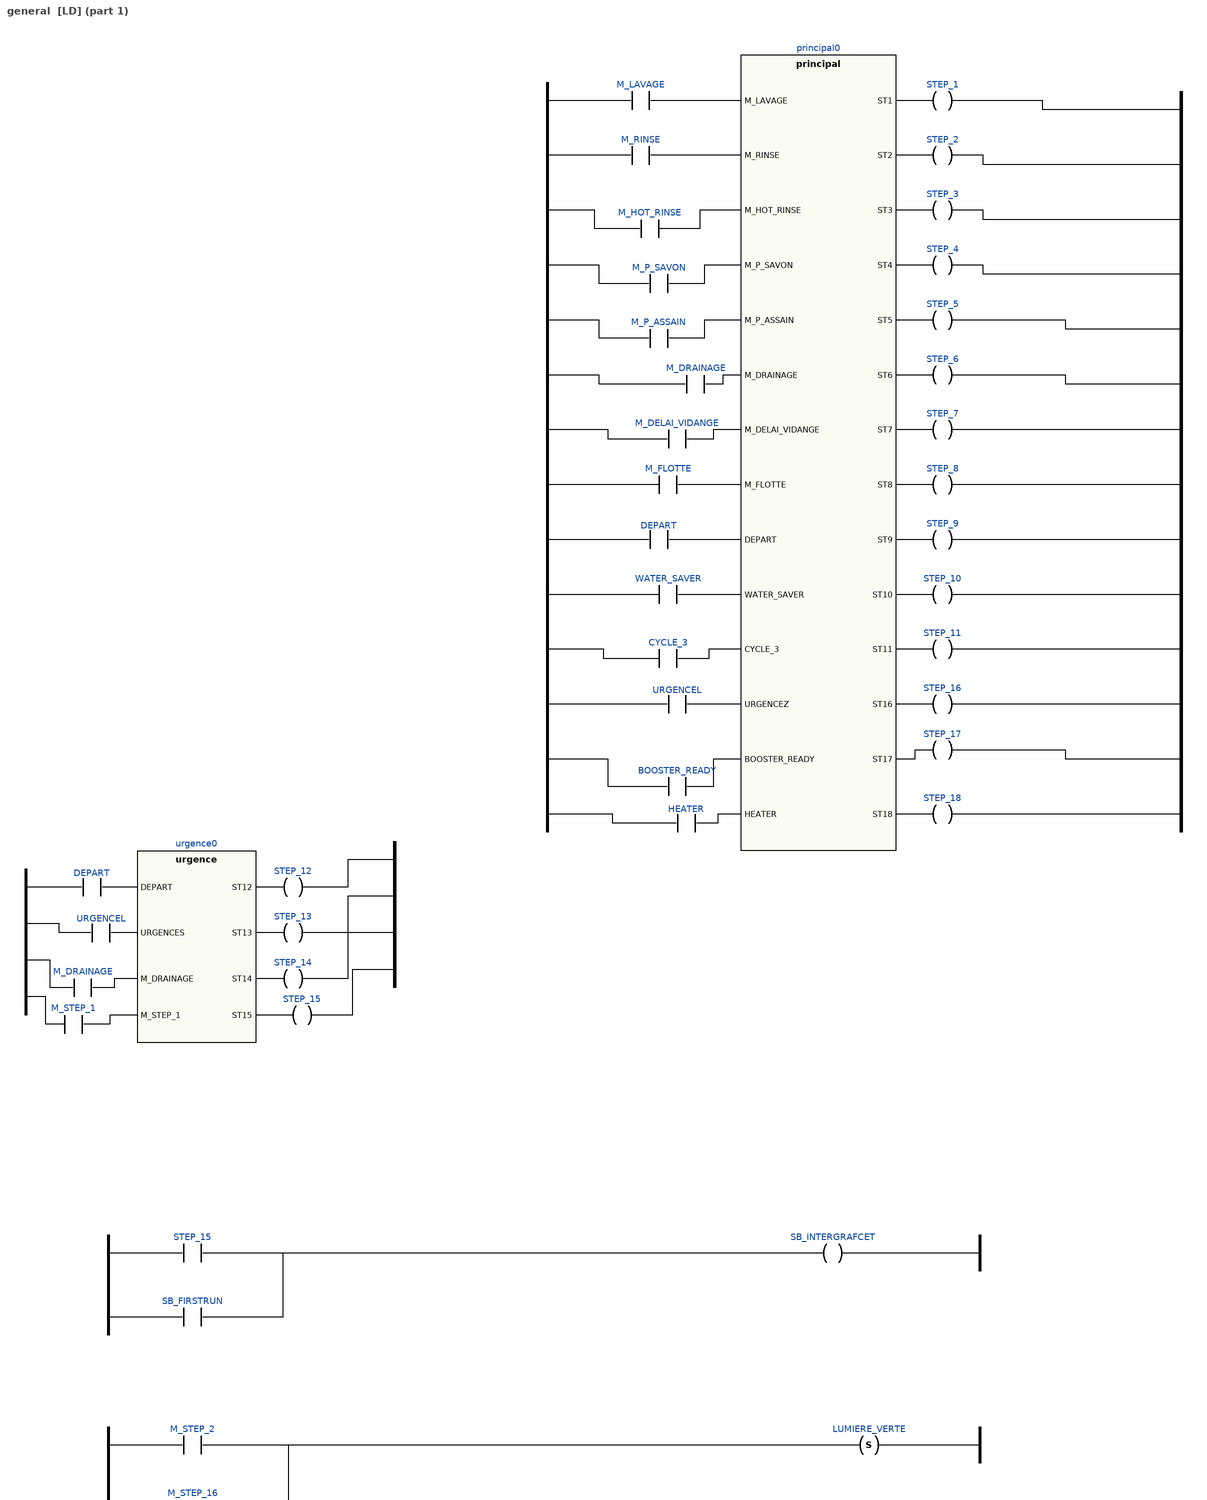
(* LD diagram, written out as Structured Text *)
principal0(M_LAVAGE := M_LAVAGE, M_RINSE := M_RINSE, M_HOT_RINSE := M_HOT_RINSE, M_P_SAVON := M_P_SAVON, M_P_ASSAIN := M_P_ASSAIN, M_DRAINAGE := M_DRAINAGE, M_DELAI_VIDANGE := M_DELAI_VIDANGE, M_FLOTTE := M_FLOTTE, DEPART := DEPART, WATER_SAVER := WATER_SAVER, CYCLE_3 := CYCLE_3, URGENCEZ := URGENCEL, BOOSTER_READY := BOOSTER_READY, HEATER := HEATER);
STEP_1 := principal0.ST1;
STEP_2 := principal0.ST2;
STEP_3 := principal0.ST3;
STEP_4 := principal0.ST4;
STEP_5 := principal0.ST5;
STEP_6 := principal0.ST6;
STEP_7 := principal0.ST7;
STEP_8 := principal0.ST8;
STEP_9 := principal0.ST9;
STEP_10 := principal0.ST10;
STEP_11 := principal0.ST11;
STEP_16 := principal0.ST16;
STEP_17 := principal0.ST17;
STEP_18 := principal0.ST18;
urgence0(DEPART := DEPART, URGENCES := URGENCEL, M_DRAINAGE := M_DRAINAGE, M_STEP_1 := M_STEP_1);
STEP_12 := urgence0.ST12;
STEP_13 := urgence0.ST13;
STEP_14 := urgence0.ST14;
STEP_15 := urgence0.ST15;
SB_INTERGRAFCET := STEP_15 OR SB_FIRSTRUN;
IF M_STEP_2 OR M_STEP_16 THEN LUMIERE_VERTE := TRUE; END_IF;
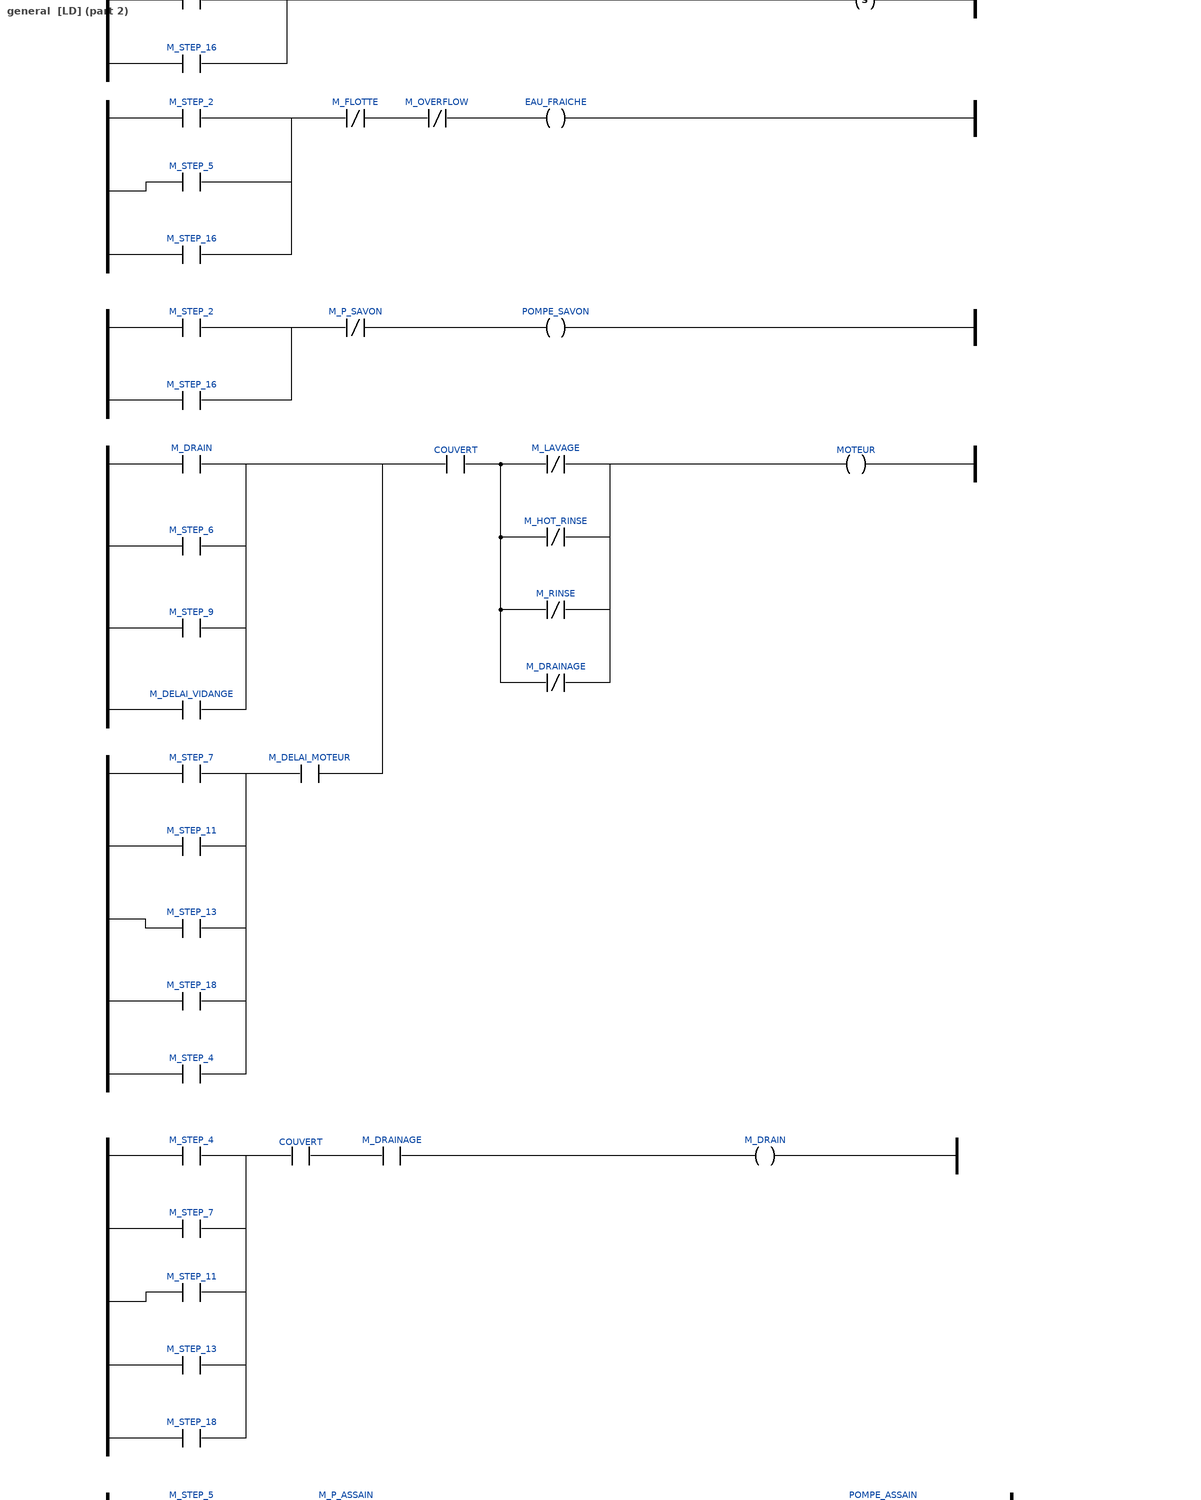
EAU_FRAICHE := (M_STEP_2 OR M_STEP_5 OR M_STEP_16) AND NOT M_FLOTTE AND NOT M_OVERFLOW;
POMPE_SAVON := (M_STEP_2 OR M_STEP_16) AND NOT M_P_SAVON;
MOTEUR := (M_DRAIN OR M_STEP_6 OR M_STEP_9 OR M_DELAI_VIDANGE OR (M_STEP_7 OR M_STEP_11 OR M_STEP_13 OR M_STEP_18 OR M_STEP_4) AND M_DELAI_MOTEUR) AND COUVERT AND (NOT M_LAVAGE OR NOT M_HOT_RINSE OR NOT M_RINSE OR NOT M_DRAINAGE);
M_DRAIN := (M_STEP_4 OR M_STEP_7 OR M_STEP_11 OR M_STEP_13 OR M_STEP_18) AND COUVERT AND M_DRAINAGE;
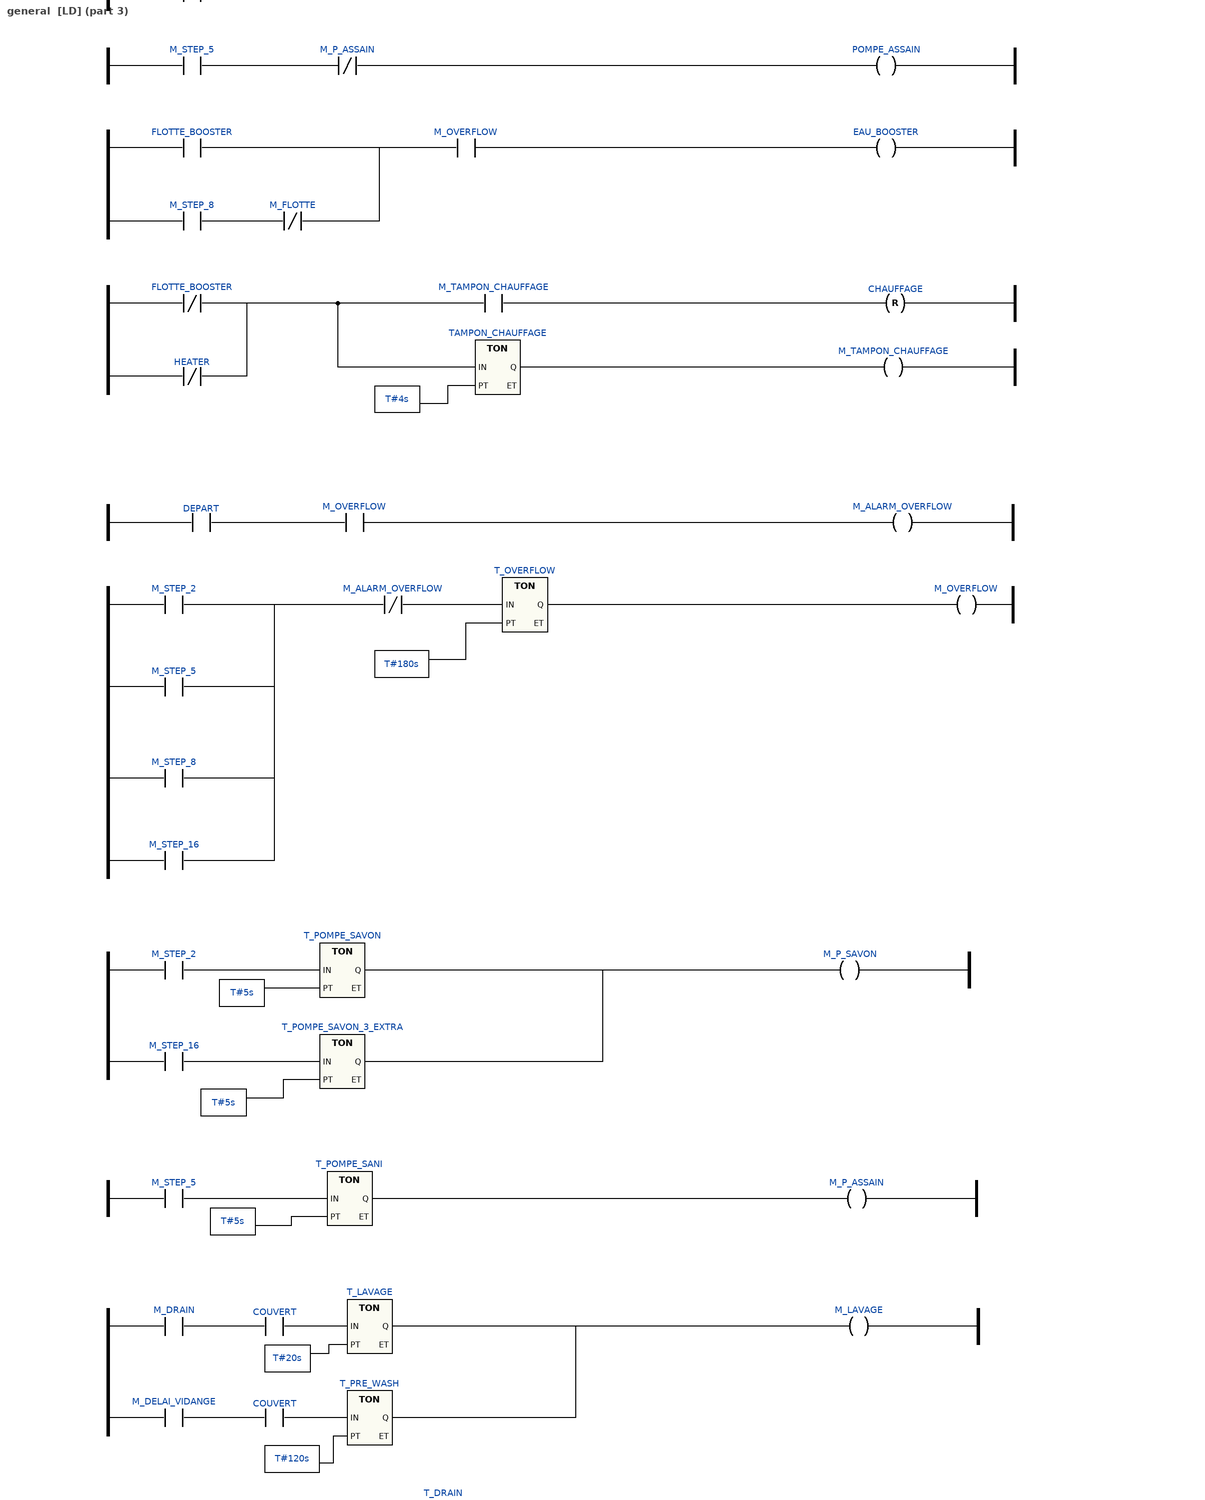
POMPE_ASSAIN := M_STEP_5 AND NOT M_P_ASSAIN;
EAU_BOOSTER := (M_STEP_8 AND NOT M_FLOTTE OR FLOTTE_BOOSTER) AND M_OVERFLOW;
IF (NOT FLOTTE_BOOSTER OR NOT HEATER) AND M_TAMPON_CHAUFFAGE THEN CHAUFFAGE := FALSE; END_IF;
TAMPON_CHAUFFAGE(IN := NOT FLOTTE_BOOSTER, PT := T#4s);
M_TAMPON_CHAUFFAGE := TAMPON_CHAUFFAGE.Q;
M_ALARM_OVERFLOW := DEPART AND M_OVERFLOW;
T_OVERFLOW(IN := (M_STEP_2 OR M_STEP_5 OR M_STEP_8 OR M_STEP_16) AND NOT M_ALARM_OVERFLOW, PT := T#180s);
M_OVERFLOW := T_OVERFLOW.Q;
T_POMPE_SAVON(IN := M_STEP_2, PT := T#5s);
T_POMPE_SAVON_3_EXTRA(IN := M_STEP_16, PT := T#5s);
M_P_SAVON := T_POMPE_SAVON.Q OR T_POMPE_SAVON_3_EXTRA.Q;
T_POMPE_SANI(IN := M_STEP_5, PT := T#5s);
M_P_ASSAIN := T_POMPE_SANI.Q;
T_LAVAGE(IN := M_DRAIN AND COUVERT, PT := T#20s);
T_PRE_WASH(IN := M_DELAI_VIDANGE AND COUVERT, PT := T#120s);
M_LAVAGE := T_LAVAGE.Q OR T_PRE_WASH.Q;
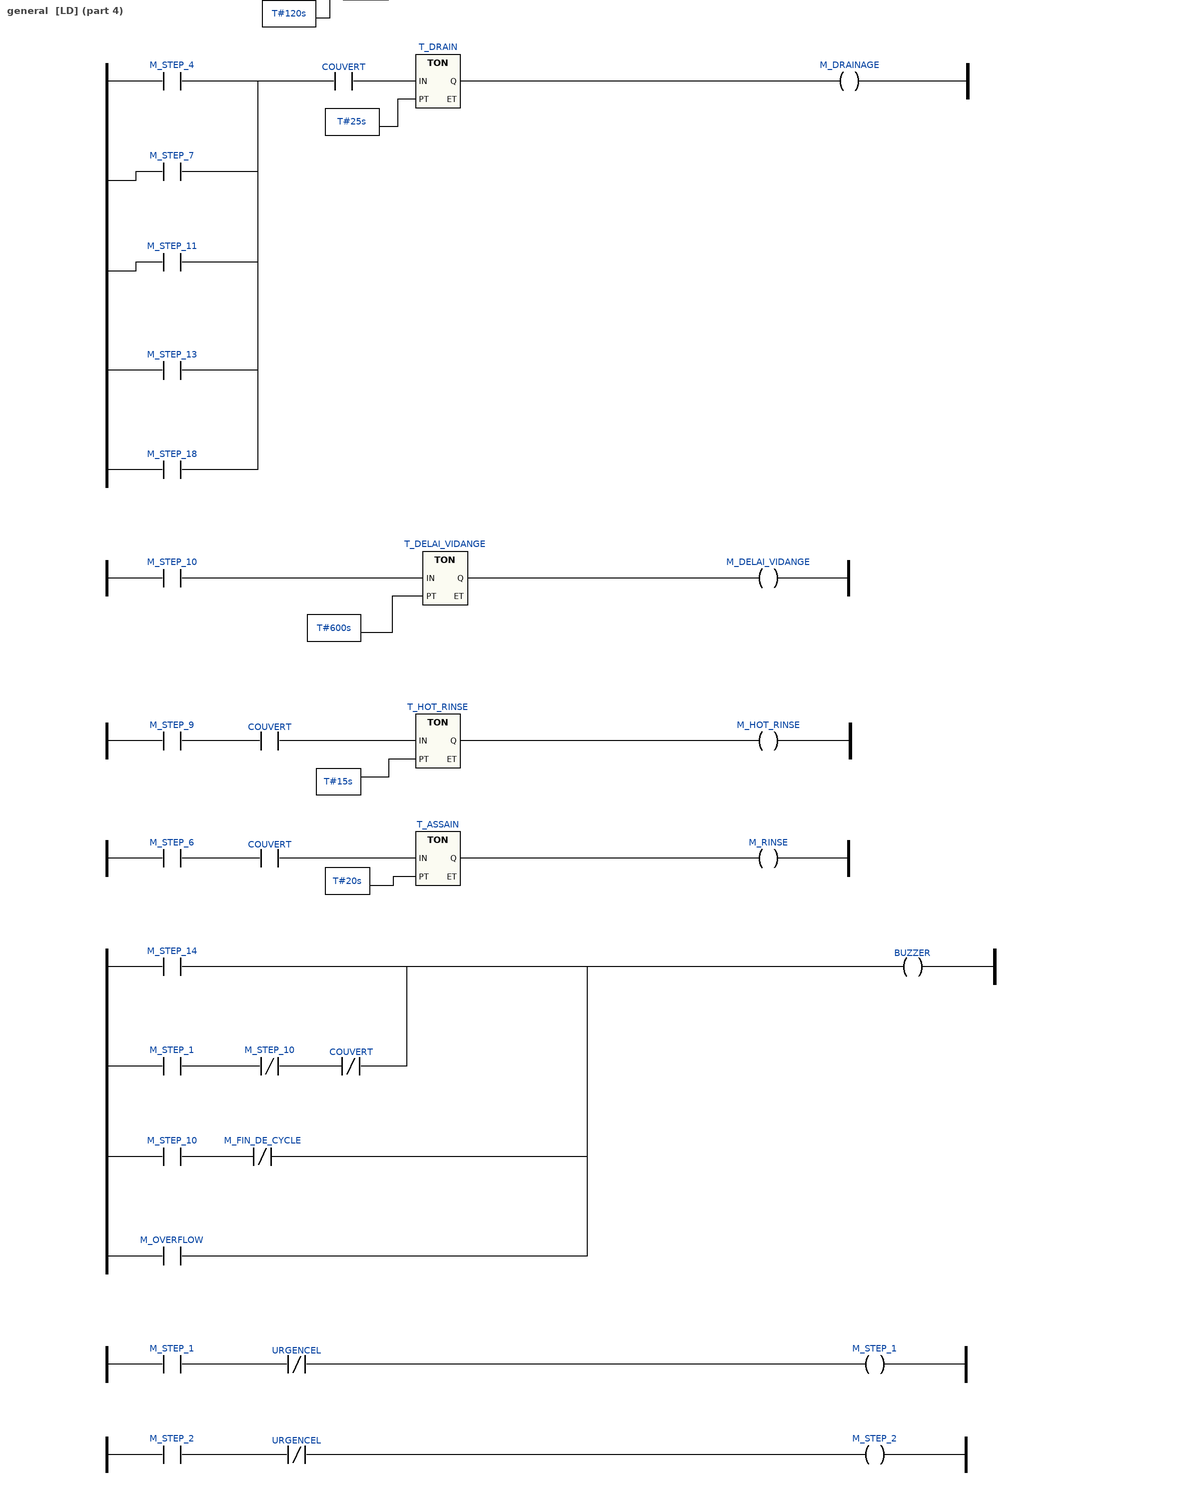
T_DRAIN(IN := (M_STEP_4 OR M_STEP_7 OR M_STEP_11 OR M_STEP_13 OR M_STEP_18) AND COUVERT, PT := T#25s);
M_DRAINAGE := T_DRAIN.Q;
T_DELAI_VIDANGE(IN := M_STEP_10, PT := T#600s);
M_DELAI_VIDANGE := T_DELAI_VIDANGE.Q;
T_HOT_RINSE(IN := M_STEP_9 AND COUVERT, PT := T#15s);
M_HOT_RINSE := T_HOT_RINSE.Q;
T_ASSAIN(IN := M_STEP_6 AND COUVERT, PT := T#20s);
M_RINSE := T_ASSAIN.Q;
BUZZER := M_STEP_14 OR M_STEP_1 AND NOT M_STEP_10 AND NOT COUVERT OR M_STEP_10 AND NOT M_FIN_DE_CYCLE OR M_OVERFLOW;
M_STEP_1 := M_STEP_1 AND NOT URGENCEL;
M_STEP_2 := M_STEP_2 AND NOT URGENCEL;
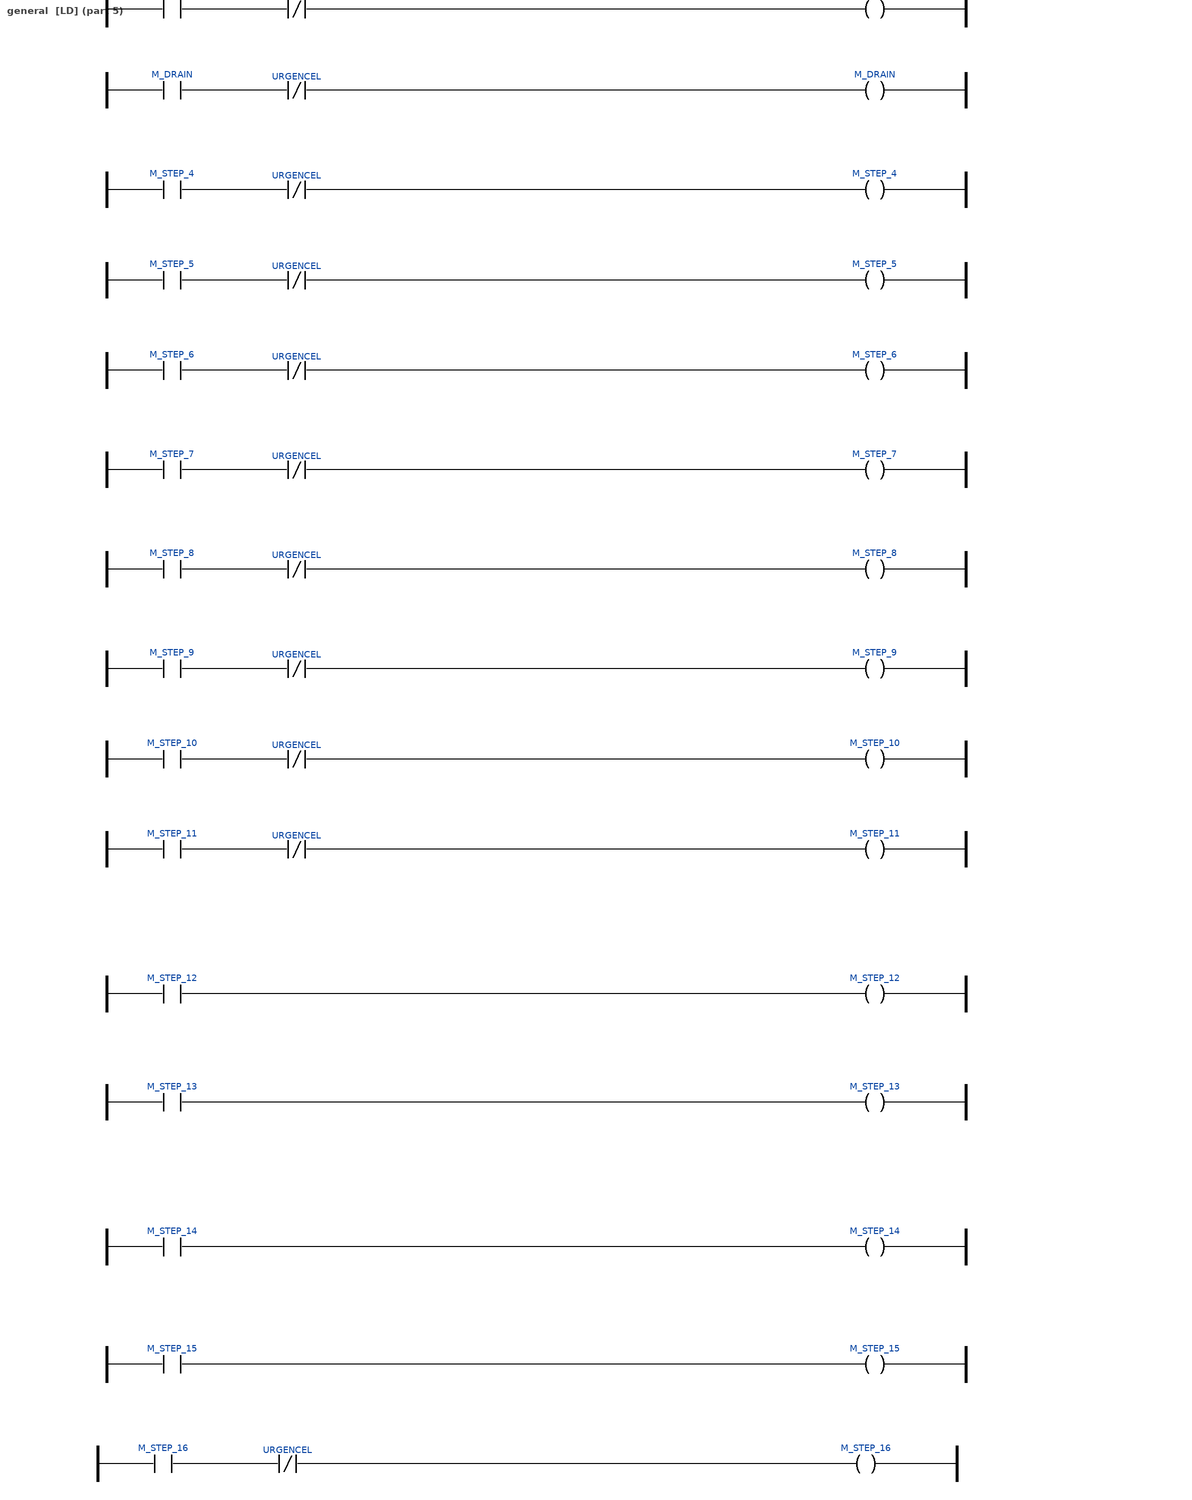
M_DRAIN := M_DRAIN AND NOT URGENCEL;
M_STEP_4 := M_STEP_4 AND NOT URGENCEL;
M_STEP_5 := M_STEP_5 AND NOT URGENCEL;
M_STEP_6 := M_STEP_6 AND NOT URGENCEL;
M_STEP_7 := M_STEP_7 AND NOT URGENCEL;
M_STEP_8 := M_STEP_8 AND NOT URGENCEL;
M_STEP_9 := M_STEP_9 AND NOT URGENCEL;
M_STEP_10 := M_STEP_10 AND NOT URGENCEL;
M_STEP_11 := M_STEP_11 AND NOT URGENCEL;
M_STEP_12 := M_STEP_12;
M_STEP_13 := M_STEP_13;
M_STEP_14 := M_STEP_14;
M_STEP_15 := M_STEP_15;
M_STEP_16 := M_STEP_16 AND NOT URGENCEL;
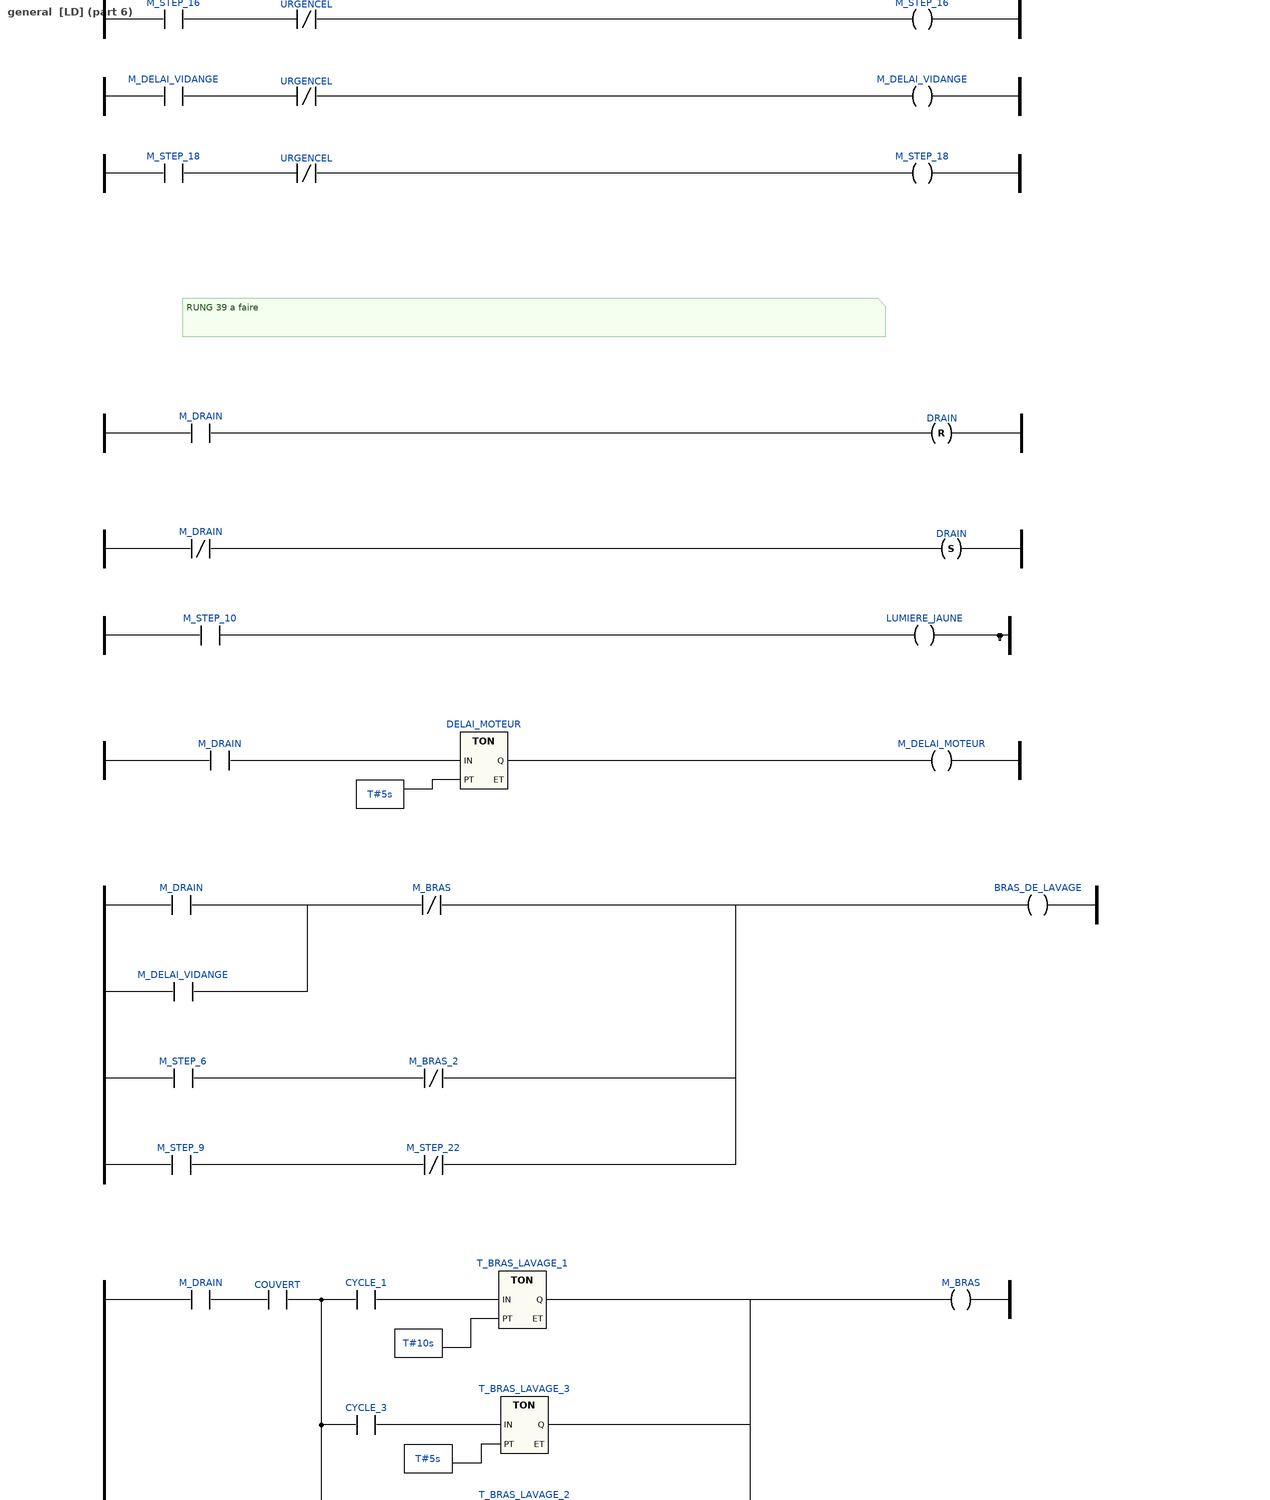
M_DELAI_VIDANGE := M_DELAI_VIDANGE AND NOT URGENCEL;
M_STEP_18 := M_STEP_18 AND NOT URGENCEL;
(* RUNG 39 a faire *)
IF M_DRAIN THEN DRAIN := FALSE; END_IF;
IF NOT M_DRAIN THEN DRAIN := TRUE; END_IF;
LUMIERE_JAUNE := M_STEP_10;
DELAI_MOTEUR(IN := M_DRAIN, PT := T#5s);
M_DELAI_MOTEUR := DELAI_MOTEUR.Q;
BRAS_DE_LAVAGE := (M_DRAIN OR M_DELAI_VIDANGE) AND NOT M_BRAS OR M_STEP_6 AND NOT M_BRAS_2 OR M_STEP_9 AND NOT M_STEP_22;
T_BRAS_LAVAGE_1(IN := M_DRAIN AND COUVERT AND CYCLE_1, PT := T#10s);
T_BRAS_LAVAGE_3(IN := M_DRAIN AND COUVERT AND CYCLE_3, PT := T#5s);
T_BRAS_LAVAGE_2(IN := M_DRAIN AND COUVERT AND NOT CYCLE_1 AND NOT CYCLE_3, PT := T#40s);
T_BRAS_PRE_LAVAGE_3(IN := M_DELAI_VIDANGE AND COUVERT AND CYCLE_3, PT := T#30s);
M_BRAS := T_BRAS_LAVAGE_1.Q OR T_BRAS_LAVAGE_3.Q OR T_BRAS_LAVAGE_2.Q OR T_BRAS_PRE_LAVAGE_3.Q;
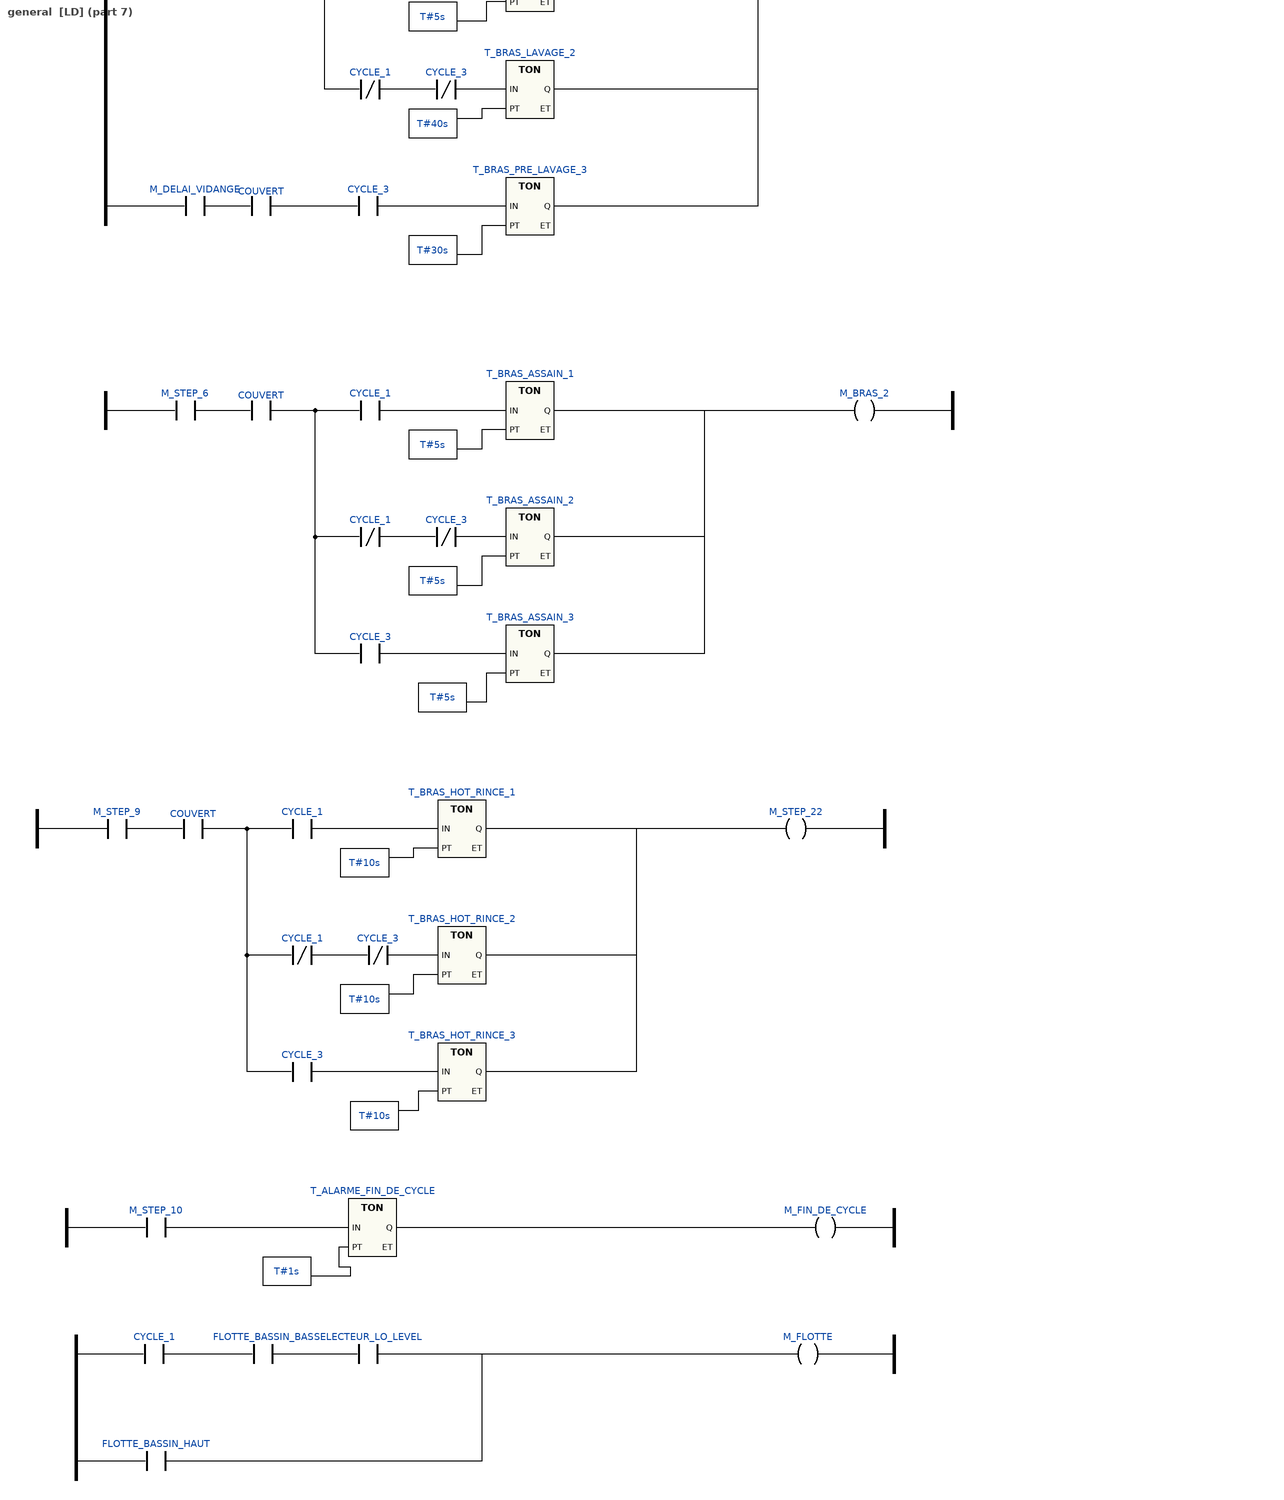
T_BRAS_ASSAIN_1(IN := M_STEP_6 AND COUVERT AND CYCLE_1, PT := T#5s);
T_BRAS_ASSAIN_2(IN := M_STEP_6 AND COUVERT AND NOT CYCLE_1 AND NOT CYCLE_3, PT := T#5s);
T_BRAS_ASSAIN_3(IN := M_STEP_6 AND COUVERT AND CYCLE_3, PT := T#5s);
M_BRAS_2 := T_BRAS_ASSAIN_1.Q OR T_BRAS_ASSAIN_2.Q OR T_BRAS_ASSAIN_3.Q;
T_BRAS_HOT_RINCE_1(IN := M_STEP_9 AND COUVERT AND CYCLE_1, PT := T#10s);
T_BRAS_HOT_RINCE_2(IN := M_STEP_9 AND COUVERT AND NOT CYCLE_1 AND NOT CYCLE_3, PT := T#10s);
T_BRAS_HOT_RINCE_3(IN := M_STEP_9 AND COUVERT AND CYCLE_3, PT := T#10s);
M_STEP_22 := T_BRAS_HOT_RINCE_1.Q OR T_BRAS_HOT_RINCE_2.Q OR T_BRAS_HOT_RINCE_3.Q;
T_ALARME_FIN_DE_CYCLE(IN := M_STEP_10, PT := T#1s);
M_FIN_DE_CYCLE := T_ALARME_FIN_DE_CYCLE.Q;
M_FLOTTE := CYCLE_1 AND FLOTTE_BASSIN_BAS AND SELECTEUR_LO_LEVEL OR FLOTTE_BASSIN_HAUT;
END_PROGRAM

CONFIGURATION Config0
  RESOURCE Res0 ON PLC
    TASK task0(INTERVAL := T#20ms, PRIORITY := 0);
    PROGRAM instance0 WITH task0 : general;
  END_RESOURCE
END_CONFIGURATION
